Staubli VAL3: init.pgx

program init()
begin
  io:sToShow="程序复位，准备开始"
end
